// TIA Portal V16 export
// export: Created 2022-02-04T14:40:18.8117831Z, ExportSetting WithDefaults, DisplayName Totally Integrated Automation Portal, DisplayVersion V16 Update 1, DisplayName TIA Portal Version Control Interface, DisplayVersion V16, DisplayName TIA Portal Openness, DisplayVersion V16, DisplayName SINAMICS Startdrive Advanced, DisplayVersion V16 Update 5, DisplayName SINAMICS Startdrive G130, G150, S120, S150, SINAMICS MV, S210, DisplayVersion V16 Update 5, DisplayName SINAMICS Startdrive G110M, G120, G120C, G120D, G120P, G115D, DisplayVersion V16 Update 5, DisplayName STEP 7 Professional, DisplayVersion V16, DisplayName STEP 7 Safety, DisplayVersion V16, DisplayName WinCC Advanced, DisplayVersion V16, DisplayName SIMATIC Visualization Architect, DisplayVersion V16
DATA_BLOCK "IM"   // DB10
VERSION : 0.1
// stored: AutoNumber true, InstanceOfName FB_IM, InstanceOfType FB
"FB_IM"
   // VAR RETAIN
   //    M_211_Load_Transp { S7_SetPoint := 'True'} : "FB_IM2x1";
   //    M_311_Strip_Remov { S7_SetPoint := 'True'} : "FB_IM1x1";
   //    M_212_Sort_Elevator { S7_SetPoint := 'True'} : "FB_IM2x2S";
   //    M_213_ConvElevator { S7_SetPoint := 'True'} : "FB_IM1x1";
   //    M_222_Main_Sort_Slide { S7_SetPoint := 'True'} : "FB_IM1x1";
   //    M_325_Tr_Hill { S7_SetPoint := 'True'} : "FB_IM1x1";
   //    M_223_Evaluation_area { S7_SetPoint := 'True'} : "FB_IM1x1";
   //    M_224_Individ_dispensing { S7_SetPoint := 'True'} : "FB_IM2x2S";
   //    M_225_Conveyor_with_lugs { S7_SetPoint := 'True'} : "FB_IM1x1";
   //    M_235_Movable_board { S7_SetPoint := 'True'} : "FB_IM2x2S";
   //    M_231_Roller_conveyor { S7_SetPoint := 'True'} : "FB_IM1x1";
   //    M_323_Small_Chain { S7_SetPoint := 'True'} : "FB_IM1x1";
   //    M_214_Gasket_receiver { S7_SetPoint := 'True'} : "FB_IM1x1";
   //    M_312_First_slide { S7_SetPoint := 'True'} : "FB_IM1x1";
   //    M_313_AF_slide_conv { S7_SetPoint := 'True'} : "FB_IM1x1";
   //    M_316_Padloader_IN2 { S7_SetPoint := 'True'} : "FB_IM1x1";
   //    M_314_Second_slide { S7_SetPoint := 'True'} : "FB_IM1x1";
   //    M_315_Third_slide { S7_SetPoint := 'True'} : "FB_IM1x1";
   //    M_234_Carousel_loader { S7_SetPoint := 'True'} : "FB_IM1x1";
   //    M_330_Scrap_Conv { S7_SetPoint := 'True'} : "FB_IM1x1";
   //    M_331_Scrap_conveyor { S7_SetPoint := 'True'} : "FB_IM1x1";
   //    M_332_Dump_lug_conv { S7_SetPoint := 'True'} : "FB_IM1x1";
   //    M_333_Defective_roller { S7_SetPoint := 'True'} : "FB_IM1x1";
   //    M_334_Layer_set_conv { S7_SetPoint := 'True'} : "FB_IM1x1";
   //    M_335_Lay_fork_scrap { S7_SetPoint := 'True'} : "FB_IM2x2";
   //    M_336_PFM_elevator { S7_SetPoint := 'True'} : "FB_IM2x2S";
   // END_VAR
BEGIN
END_DATA_BLOCK
